{attribute addProperty BoxType "EL2212-0000-0020"}
{attribute addProperty Id "ControlAT %Q*Control_689B20B6162"}
{attribute addProperty CRC "150882576"}
{attribute addProperty SizeInBites "16"}
{attribute addProperty SizeInBytes "2"}
TYPE DOX_Control_Channel_08FE4910 :
STRUCT
	{attribute addProperty Name "Control"}
	Control AT %Q* : Control_689B20B6;
END_STRUCT
END_TYPE

(* stored: Version 1.2.0.0, ProductVersion 3.1.4024.9
   DUT DOX_Control_Channel_08FE4910: Id {0127be6d-6727-4c54-8f47-a043e0c5cbcf} *)
